Fanuc KAREL source: kd00076.KL

-- PROVISIONAL review KL for V770-1; original PC SHA256 38b1d0f184bf5f9aa531995b9c0e21e2e1cbbdd3ac5463d8aae09812cbca844a
-- Incomplete behavior may be omitted. Consult companion uncertainty JSON. Do not deploy.
PROGRAM KD00076
%NOLOCKGROUP
VAR
  I : INTEGER
  J : INTEGER
  B : BOOLEAN
  R : REAL
  S : STRING[80]
BEGIN
  -- UNRESOLVED_PC offsets 5-7; opcodes 9D,3C
  -- UNRESOLVED_PC offsets 12-16; opcodes 7F
END KD00076
